// The two CV values map a Boolean demand into engineering output units.
TYPE ST_BangBang_Cfg :
STRUCT
    hysteresis : ST_Hysteresis_Cfg;
    lowValue   : REAL := 0.0;
    highValue  : REAL := 100.0;
END_STRUCT
END_TYPE

(* stored: Version 1.1.0.1, ProductVersion 3.1.4026.12
   DUT ST_BangBang_Cfg: Id {5e1b4e16-9ba8-424b-8e19-255dd6b0580c} *)
